// TIA Portal project "SELECTOR" (V16)

(* hardware
DEVICE "S7-1200 station_1"  S7-1200 Station
   slot 0: "Rack_0"  S7-1200 Rack  Rack  V1.0
   slot 1: "PLC_1"  CPU 1212C AC/DC/Rly  6ES7 212-1BE40-0XB0  V4.0
*)

// ===== PLC "PLC_1"  CPU 1212C AC/DC/Rly =====

VAR_GLOBAL   // PLC tag table "Default tag table"
   "START 1" AT %I0.2 : Bool;
   "START 2" AT %I0.4 : Bool;
   "STOP" AT %I0.3 : Bool;
   "MANUAL" AT %I0.5 : Bool;
   "AUTOMATIC" AT %I0.6 : Bool;
   "COIL 1" AT %Q0.0 : Bool;
   "COIL 2" AT %Q0.1 : Bool;
   "COIL 3" AT %Q0.2 : Bool;
   "COIL 4" AT %Q0.3 : Bool;
   "M1" AT %M0.0 : Bool;
   "M2" AT %M0.1 : Bool;
   "M3" AT %M0.2 : Bool;
   "M4" AT %M0.3 : Bool;
   "M5" AT %M0.4 : Bool;
   "M6" AT %M0.5 : Bool;
   "M7" AT %M0.6 : Bool;
   "M8" AT %M0.7 : Bool;
   "M9" AT %M1.0 : Bool;
   "M10" AT %M1.1 : Bool;
   "M11" AT %M1.2 : Bool;
   "M12" AT %M1.3 : Bool;
   "M13" AT %M1.4 : Bool;
END_VAR

// folder: System blocks/Program resources

DATA_BLOCK "T1"   // DB1
{ S7_Optimized_Access := 'TRUE' }
AUTHOR : Simatic
FAMILY : IEC
NAME : IEC_TMR
VERSION : 1.0
// stored: InstanceOfName IEC_TIMER
"IEC_TIMER"
BEGIN
END_DATA_BLOCK

DATA_BLOCK "T2"   // DB2
{ S7_Optimized_Access := 'TRUE' }
AUTHOR : Simatic
FAMILY : IEC
NAME : IEC_TMR
VERSION : 1.0
// stored: InstanceOfName IEC_TIMER
"IEC_TIMER"
BEGIN
END_DATA_BLOCK

DATA_BLOCK "T3"   // DB3
{ S7_Optimized_Access := 'TRUE' }
AUTHOR : Simatic
FAMILY : IEC
NAME : IEC_TMR
VERSION : 1.0
// stored: InstanceOfName IEC_TIMER
"IEC_TIMER"
BEGIN
END_DATA_BLOCK

DATA_BLOCK "T4"   // DB4
{ S7_Optimized_Access := 'TRUE' }
AUTHOR : Simatic
FAMILY : IEC
NAME : IEC_TMR
VERSION : 1.0
// stored: InstanceOfName IEC_TIMER
"IEC_TIMER"
BEGIN
END_DATA_BLOCK

DATA_BLOCK "T5"   // DB5
{ S7_Optimized_Access := 'TRUE' }
AUTHOR : Simatic
FAMILY : IEC
NAME : IEC_TMR
VERSION : 1.0
// stored: InstanceOfName IEC_TIMER
"IEC_TIMER"
BEGIN
END_DATA_BLOCK

// folder: (top level)

ORGANIZATION_BLOCK "Main"   // OB1, LAD, ProgramCycle
TITLE = "Main Program Sweep (Cycle)"
{ S7_Optimized_Access := 'TRUE' }
VERSION : 0.1
   VAR_INPUT
      Initial_Call : Bool;   // Initial call of this OB
      Remanence : Bool;   // =True, if remanent data are available
   END_VAR
   VAR_TEMP   // added for the SCL form of the ladder/FBD networks
      _w1 : Bool;
   END_VAR
BEGIN

REGION Network 1
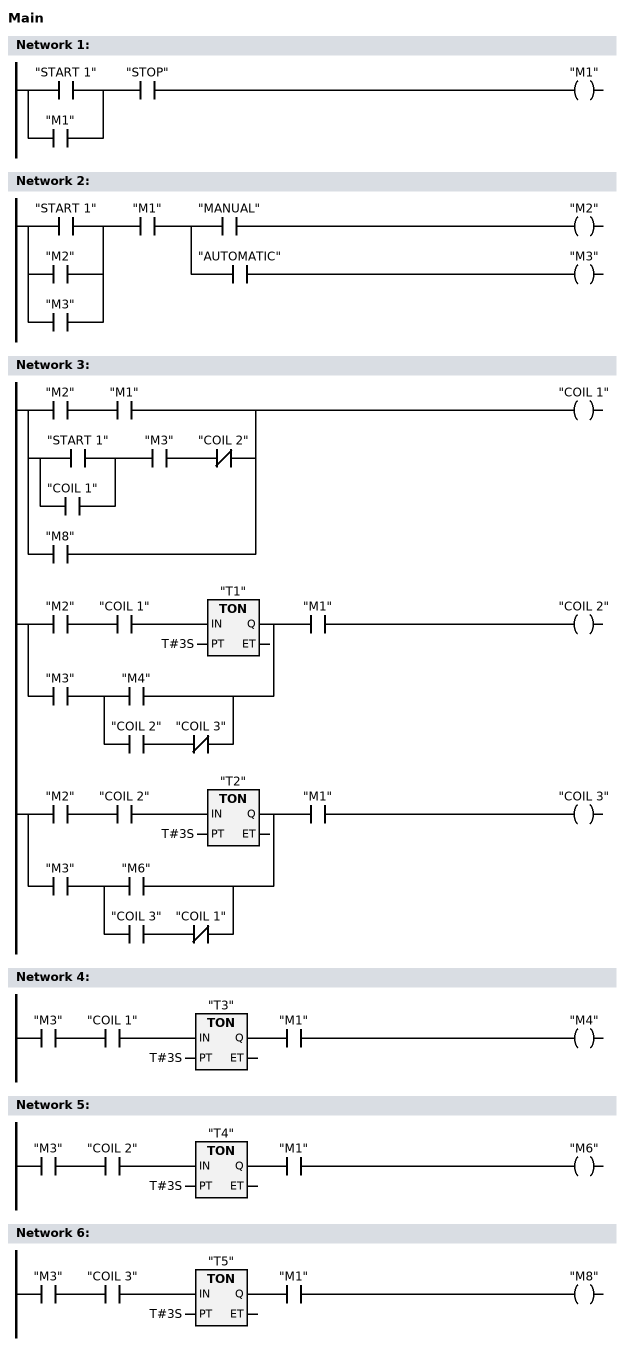
   RUNG wire#powerrail
      Contact( "START 1" )
      wire#w1
      Contact( "STOP" )
      Coil( "M1" )
   END_RUNG
   RUNG wire#powerrail
      Contact( "M1" )
   END_RUNG wire#w1
   // the same network as SCL:
   "M1" := ("START 1" OR "M1") AND "STOP";
END_REGION

REGION Network 2
   RUNG wire#powerrail
      Contact( "START 1" )
      wire#w1
      Contact( "M1" )
      wire#w2
      Contact( "MANUAL" )
      Coil( "M2" )
   END_RUNG
   RUNG wire#powerrail
      Contact( "M2" )
   END_RUNG wire#w1
   RUNG wire#powerrail
      Contact( "M3" )
   END_RUNG wire#w1
   RUNG wire#w2
      Contact( "AUTOMATIC" )
      Coil( "M3" )
   END_RUNG
   // the same network as SCL:
   #_w1 := ("START 1" OR "M2" OR "M3") AND "M1";
   "M2" := #_w1 AND "MANUAL";
   "M3" := #_w1 AND "AUTOMATIC";
END_REGION

REGION Network 3
   "COIL 1" := ("M2" AND "M1") OR (("START 1" OR "COIL 1") AND "M3" AND NOT "COIL 2") OR "M8";
   "T1".TON(IN := "M2" AND "COIL 1", PT := T#3S);
   "COIL 2" := ("T1".Q OR ("M3" AND ("M4" OR ("COIL 2" AND NOT "COIL 3")))) AND "M1";
   "T2".TON(IN := "M2" AND "COIL 2", PT := T#3S);
   "COIL 3" := ("T2".Q OR ("M3" AND ("M6" OR ("COIL 3" AND NOT "COIL 1")))) AND "M1";
END_REGION

REGION Network 4
   "T3".TON(IN := "M3" AND "COIL 1", PT := T#3S);
   "M4" := "T3".Q AND "M1";
END_REGION

REGION Network 5
   "T4".TON(IN := "M3" AND "COIL 2", PT := T#3S);
   "M6" := "T4".Q AND "M1";
END_REGION

REGION Network 6
   "T5".TON(IN := "M3" AND "COIL 3", PT := T#3S);
   "M8" := "T5".Q AND "M1";
END_REGION
END_ORGANIZATION_BLOCK